// TIA Portal project "LabPLC" (V13)

(* hardware
DEVICE "S7-1200 station_1"  S7-1200 Station
   slot 0: "Rack_0"  Rack  V1.0
   slot 1: "LabPLC"  CPU 1215C DC/DC/DC  6ES7 215-1AG40-0XB0  V4.0
*)

// ===== PLC "LabPLC"  CPU 1215C DC/DC/DC =====

VAR_GLOBAL   // PLC tag table "Default tag table"
   "iTemp" AT %MW100 : Int;
   "PWM_Q1" AT %QW1002 : Int;
   "AxisFrequency_Pulse" AT %Q0.1 : Bool;
END_VAR

TYPE "User_data_type_1"
   STRUCT
      Notes : Array[0..15000] of Byte;
   END_STRUCT;
END_TYPE

DATA_BLOCK "dbInsMaster"   // DB2
{ S7_Optimized_Access := 'FALSE' }
VERSION : 0.1
// stored: InstanceOfName fbMaster
"fbMaster"
BEGIN
END_DATA_BLOCK

DATA_BLOCK "dbToneToFrequency"   // DB3
{ S7_Optimized_Access := 'FALSE' }
VERSION : 0.1
   VAR
      Freq : Array[0..128] of Int;
   END_VAR
BEGIN
   Freq[0] := 8;
   Freq[1] := 9;
   Freq[2] := 9;
   Freq[3] := 10;
   Freq[4] := 10;
   Freq[5] := 11;
   Freq[6] := 12;
   Freq[7] := 12;
   Freq[8] := 13;
   Freq[9] := 14;
   Freq[10] := 15;
   Freq[11] := 15;
   Freq[12] := 16;
   Freq[13] := 17;
   Freq[14] := 18;
   Freq[15] := 19;
   Freq[16] := 21;
   Freq[17] := 22;
   Freq[18] := 23;
   Freq[19] := 24;
   Freq[20] := 26;
   Freq[21] := 28;
   Freq[22] := 29;
   Freq[23] := 31;
   Freq[24] := 33;
   Freq[25] := 35;
   Freq[26] := 37;
   Freq[27] := 39;
   Freq[28] := 41;
   Freq[29] := 44;
   Freq[30] := 46;
   Freq[31] := 49;
   Freq[32] := 52;
   Freq[33] := 55;
   Freq[34] := 58;
   Freq[35] := 62;
   Freq[36] := 65;
   Freq[37] := 69;
   Freq[38] := 73;
   Freq[39] := 78;
   Freq[40] := 82;
   Freq[41] := 87;
   Freq[42] := 92;
   Freq[43] := 98;
   Freq[44] := 104;
   Freq[45] := 110;
   Freq[46] := 117;
   Freq[47] := 123;
   Freq[48] := 131;
   Freq[49] := 139;
   Freq[50] := 147;
   Freq[51] := 156;
   Freq[52] := 165;
   Freq[53] := 175;
   Freq[54] := 185;
   Freq[55] := 196;
   Freq[56] := 208;
   Freq[57] := 220;
   Freq[58] := 233;
   Freq[59] := 247;
   Freq[60] := 262;
   Freq[61] := 277;
   Freq[62] := 294;
   Freq[63] := 311;
   Freq[64] := 330;
   Freq[65] := 349;
   Freq[66] := 370;
   Freq[67] := 392;
   Freq[68] := 415;
   Freq[69] := 440;
   Freq[70] := 466;
   Freq[71] := 494;
   Freq[72] := 523;
   Freq[73] := 554;
   Freq[74] := 587;
   Freq[75] := 622;
   Freq[76] := 659;
   Freq[77] := 698;
   Freq[78] := 740;
   Freq[79] := 784;
   Freq[80] := 831;
   Freq[81] := 880;
   Freq[82] := 932;
   Freq[83] := 988;
   Freq[84] := 1047;
   Freq[85] := 1109;
   Freq[86] := 1175;
   Freq[87] := 1245;
   Freq[88] := 1319;
   Freq[89] := 1397;
   Freq[90] := 1480;
   Freq[91] := 1568;
   Freq[92] := 1661;
   Freq[93] := 1760;
   Freq[94] := 1865;
   Freq[95] := 1976;
   Freq[96] := 2093;
   Freq[97] := 2217;
   Freq[98] := 2349;
   Freq[99] := 2489;
   Freq[100] := 2637;
   Freq[101] := 2794;
   Freq[102] := 2960;
   Freq[103] := 3136;
   Freq[104] := 3322;
   Freq[105] := 3520;
   Freq[106] := 3729;
   Freq[107] := 3951;
   Freq[108] := 4186;
   Freq[109] := 4435;
   Freq[110] := 4699;
   Freq[111] := 4978;
   Freq[112] := 5274;
   Freq[113] := 5588;
   Freq[114] := 5920;
   Freq[115] := 6272;
   Freq[116] := 6645;
   Freq[117] := 7040;
   Freq[118] := 7459;
   Freq[119] := 7902;
   Freq[120] := 8372;
   Freq[121] := 8870;
   Freq[122] := 9397;
   Freq[123] := 9956;
   Freq[124] := 10548;
   Freq[125] := 11175;
   Freq[126] := 11840;
   Freq[127] := 12544;
   Freq[128] := 13290;
END_DATA_BLOCK

DATA_BLOCK "dbTunes"   // DB4
{ S7_Optimized_Access := 'FALSE' }
VERSION : 0.1
   VAR
      Tune_01 : Array[0..5000] of Byte;
   END_VAR
BEGIN
   Tune_01[0] := 0;
   Tune_01[1] := 36;
   Tune_01[2] := 16#0090;
   Tune_01[3] := 55;
   Tune_01[4] := 1;
   Tune_01[5] := 74;
   Tune_01[6] := 16#0080;
   Tune_01[7] := 0;
   Tune_01[8] := 242;
   Tune_01[9] := 16#0090;
   Tune_01[10] := 55;
   Tune_01[11] := 1;
   Tune_01[12] := 105;
   Tune_01[13] := 16#0080;
   Tune_01[14] := 0;
   Tune_01[15] := 232;
   Tune_01[16] := 16#0090;
   Tune_01[17] := 55;
   Tune_01[18] := 1;
   Tune_01[19] := 111;
   Tune_01[20] := 16#0080;
   Tune_01[21] := 0;
   Tune_01[22] := 202;
   Tune_01[23] := 16#0090;
   Tune_01[24] := 51;
   Tune_01[25] := 1;
   Tune_01[26] := 31;
   Tune_01[27] := 16#0080;
   Tune_01[28] := 0;
   Tune_01[29] := 147;
   Tune_01[30] := 16#0090;
   Tune_01[31] := 58;
   Tune_01[32] := 0;
   Tune_01[33] := 79;
   Tune_01[34] := 16#0080;
   Tune_01[35] := 0;
   Tune_01[36] := 69;
   Tune_01[37] := 16#0090;
   Tune_01[38] := 55;
   Tune_01[39] := 1;
   Tune_01[40] := 160;
   Tune_01[41] := 16#0080;
   Tune_01[42] := 0;
   Tune_01[43] := 165;
   Tune_01[44] := 16#0090;
   Tune_01[45] := 51;
   Tune_01[46] := 1;
   Tune_01[47] := 31;
   Tune_01[48] := 16#0080;
   Tune_01[49] := 0;
   Tune_01[50] := 169;
   Tune_01[51] := 16#0090;
   Tune_01[52] := 58;
   Tune_01[53] := 0;
   Tune_01[54] := 85;
   Tune_01[55] := 16#0080;
   Tune_01[56] := 0;
   Tune_01[57] := 51;
   Tune_01[58] := 16#0090;
   Tune_01[59] := 55;
   Tune_01[60] := 2;
   Tune_01[61] := 235;
   Tune_01[62] := 16#0080;
   Tune_01[63] := 1;
   Tune_01[64] := 166;
   Tune_01[65] := 16#0090;
   Tune_01[66] := 62;
   Tune_01[67] := 1;
   Tune_01[68] := 121;
   Tune_01[69] := 16#0080;
   Tune_01[70] := 0;
   Tune_01[71] := 216;
   Tune_01[72] := 16#0090;
   Tune_01[73] := 62;
   Tune_01[74] := 1;
   Tune_01[75] := 115;
   Tune_01[76] := 16#0080;
   Tune_01[77] := 0;
   Tune_01[78] := 208;
   Tune_01[79] := 16#0090;
   Tune_01[80] := 62;
   Tune_01[81] := 1;
   Tune_01[82] := 130;
   Tune_01[83] := 16#0080;
   Tune_01[84] := 0;
   Tune_01[85] := 223;
   Tune_01[86] := 16#0090;
   Tune_01[87] := 63;
   Tune_01[88] := 1;
   Tune_01[89] := 1;
   Tune_01[90] := 16#0080;
   Tune_01[91] := 0;
   Tune_01[92] := 165;
   Tune_01[93] := 16#0090;
   Tune_01[94] := 58;
   Tune_01[95] := 0;
   Tune_01[96] := 95;
   Tune_01[97] := 16#0080;
   Tune_01[98] := 0;
   Tune_01[99] := 69;
   Tune_01[100] := 16#0090;
   Tune_01[101] := 54;
   Tune_01[102] := 1;
   Tune_01[103] := 160;
   Tune_01[104] := 16#0080;
   Tune_01[105] := 0;
   Tune_01[106] := 156;
   Tune_01[107] := 16#0090;
   Tune_01[108] := 51;
   Tune_01[109] := 0;
   Tune_01[110] := 248;
   Tune_01[111] := 16#0080;
   Tune_01[112] := 0;
   Tune_01[113] := 176;
   Tune_01[114] := 16#0090;
   Tune_01[115] := 58;
   Tune_01[116] := 0;
   Tune_01[117] := 85;
   Tune_01[118] := 16#0080;
   Tune_01[119] := 0;
   Tune_01[120] := 79;
   Tune_01[121] := 16#0090;
   Tune_01[122] := 55;
   Tune_01[123] := 2;
   Tune_01[124] := 2;
   Tune_01[125] := 16#0080;
   Tune_01[126] := 2;
   Tune_01[127] := 143;
   Tune_01[128] := 16#0090;
   Tune_01[129] := 67;
   Tune_01[130] := 1;
   Tune_01[131] := 201;
   Tune_01[132] := 16#0080;
   Tune_01[133] := 0;
   Tune_01[134] := 131;
   Tune_01[135] := 16#0090;
   Tune_01[136] := 55;
   Tune_01[137] := 1;
   Tune_01[138] := 41;
   Tune_01[139] := 16#0080;
   Tune_01[140] := 0;
   Tune_01[141] := 161;
   Tune_01[142] := 16#0090;
   Tune_01[143] := 55;
   Tune_01[144] := 0;
   Tune_01[145] := 116;
   Tune_01[146] := 16#0080;
   Tune_01[147] := 0;
   Tune_01[148] := 34;
   Tune_01[149] := 16#0090;
   Tune_01[150] := 67;
   Tune_01[151] := 1;
   Tune_01[152] := 115;
   Tune_01[153] := 16#0080;
   Tune_01[154] := 0;
   Tune_01[155] := 164;
   Tune_01[156] := 16#0090;
   Tune_01[157] := 66;
   Tune_01[158] := 1;
   Tune_01[159] := 62;
   Tune_01[160] := 16#0080;
   Tune_01[161] := 0;
   Tune_01[162] := 153;
   Tune_01[163] := 16#0090;
   Tune_01[164] := 65;
   Tune_01[165] := 0;
   Tune_01[166] := 98;
   Tune_01[167] := 16#0080;
   Tune_01[168] := 0;
   Tune_01[169] := 49;
   Tune_01[170] := 16#0090;
   Tune_01[171] := 64;
   Tune_01[172] := 0;
   Tune_01[173] := 140;
   Tune_01[174] := 16#0080;
   Tune_01[175] := 0;
   Tune_01[176] := 6;
   Tune_01[177] := 16#0090;
   Tune_01[178] := 63;
   Tune_01[179] := 0;
   Tune_01[180] := 101;
   Tune_01[181] := 16#0080;
   Tune_01[182] := 0;
   Tune_01[183] := 45;
   Tune_01[184] := 16#0090;
   Tune_01[185] := 64;
   Tune_01[186] := 0;
   Tune_01[187] := 132;
   Tune_01[188] := 16#0080;
   Tune_01[189] := 1;
   Tune_01[190] := 212;
   Tune_01[191] := 16#0090;
   Tune_01[192] := 56;
   Tune_01[193] := 0;
   Tune_01[194] := 113;
   Tune_01[195] := 16#0080;
   Tune_01[196] := 0;
   Tune_01[197] := 183;
   Tune_01[198] := 16#0090;
   Tune_01[199] := 61;
   Tune_01[200] := 1;
   Tune_01[201] := 133;
   Tune_01[202] := 16#0080;
   Tune_01[203] := 0;
   Tune_01[204] := 198;
   Tune_01[205] := 16#0090;
   Tune_01[206] := 60;
   Tune_01[207] := 1;
   Tune_01[208] := 66;
   Tune_01[209] := 16#0080;
   Tune_01[210] := 0;
   Tune_01[211] := 118;
   Tune_01[212] := 16#0090;
   Tune_01[213] := 59;
   Tune_01[214] := 0;
   Tune_01[215] := 107;
   Tune_01[216] := 16#0080;
   Tune_01[217] := 0;
   Tune_01[218] := 45;
   Tune_01[219] := 16#0090;
   Tune_01[220] := 58;
   Tune_01[221] := 0;
   Tune_01[222] := 113;
   Tune_01[223] := 16#0080;
   Tune_01[224] := 0;
   Tune_01[225] := 20;
   Tune_01[226] := 16#0090;
   Tune_01[227] := 57;
   Tune_01[228] := 0;
   Tune_01[229] := 89;
   Tune_01[230] := 16#0080;
   Tune_01[231] := 0;
   Tune_01[232] := 60;
   Tune_01[233] := 16#0090;
   Tune_01[234] := 58;
   Tune_01[235] := 0;
   Tune_01[236] := 128;
   Tune_01[237] := 16#0080;
   Tune_01[238] := 1;
   Tune_01[239] := 213;
   Tune_01[240] := 16#0090;
   Tune_01[241] := 51;
   Tune_01[242] := 0;
   Tune_01[243] := 98;
   Tune_01[244] := 16#0080;
   Tune_01[245] := 0;
   Tune_01[246] := 192;
   Tune_01[247] := 16#0090;
   Tune_01[248] := 54;
   Tune_01[249] := 1;
   Tune_01[250] := 99;
   Tune_01[251] := 16#0080;
   Tune_01[252] := 0;
   Tune_01[253] := 245;
   Tune_01[254] := 16#0090;
   Tune_01[255] := 51;
   Tune_01[256] := 1;
   Tune_01[257] := 81;
   Tune_01[258] := 16#0080;
   Tune_01[259] := 0;
   Tune_01[260] := 104;
   Tune_01[261] := 16#0090;
   Tune_01[262] := 54;
   Tune_01[263] := 0;
   Tune_01[264] := 73;
   Tune_01[265] := 16#0080;
   Tune_01[266] := 0;
   Tune_01[267] := 89;
   Tune_01[268] := 16#0090;
   Tune_01[269] := 58;
   Tune_01[270] := 1;
   Tune_01[271] := 139;
   Tune_01[272] := 16#0080;
   Tune_01[273] := 0;
   Tune_01[274] := 164;
   Tune_01[275] := 16#0090;
   Tune_01[276] := 55;
   Tune_01[277] := 1;
   Tune_01[278] := 74;
   Tune_01[279] := 16#0080;
   Tune_01[280] := 0;
   Tune_01[281] := 110;
   Tune_01[282] := 16#0090;
   Tune_01[283] := 58;
   Tune_01[284] := 0;
   Tune_01[285] := 79;
   Tune_01[286] := 16#0080;
   Tune_01[287] := 0;
   Tune_01[288] := 79;
   Tune_01[289] := 16#0090;
   Tune_01[290] := 62;
   Tune_01[291] := 2;
   Tune_01[292] := 233;
   Tune_01[293] := 16#0080;
   Tune_01[294] := 1;
   Tune_01[295] := 144;
   Tune_01[296] := 16#0090;
   Tune_01[297] := 67;
   Tune_01[298] := 1;
   Tune_01[299] := 201;
   Tune_01[300] := 16#0080;
   Tune_01[301] := 0;
   Tune_01[302] := 131;
   Tune_01[303] := 16#0090;
   Tune_01[304] := 55;
   Tune_01[305] := 1;
   Tune_01[306] := 41;
   Tune_01[307] := 16#0080;
   Tune_01[308] := 0;
   Tune_01[309] := 161;
   Tune_01[310] := 16#0090;
   Tune_01[311] := 55;
   Tune_01[312] := 0;
   Tune_01[313] := 116;
   Tune_01[314] := 16#0080;
   Tune_01[315] := 0;
   Tune_01[316] := 34;
   Tune_01[317] := 16#0090;
   Tune_01[318] := 67;
   Tune_01[319] := 1;
   Tune_01[320] := 115;
   Tune_01[321] := 16#0080;
   Tune_01[322] := 0;
   Tune_01[323] := 164;
   Tune_01[324] := 16#0090;
   Tune_01[325] := 66;
   Tune_01[326] := 1;
   Tune_01[327] := 62;
   Tune_01[328] := 16#0080;
   Tune_01[329] := 0;
   Tune_01[330] := 153;
   Tune_01[331] := 16#0090;
   Tune_01[332] := 65;
   Tune_01[333] := 0;
   Tune_01[334] := 98;
   Tune_01[335] := 16#0080;
   Tune_01[336] := 0;
   Tune_01[337] := 49;
   Tune_01[338] := 16#0090;
   Tune_01[339] := 64;
   Tune_01[340] := 0;
   Tune_01[341] := 140;
   Tune_01[342] := 16#0080;
   Tune_01[343] := 0;
   Tune_01[344] := 6;
   Tune_01[345] := 16#0090;
   Tune_01[346] := 63;
   Tune_01[347] := 0;
   Tune_01[348] := 101;
   Tune_01[349] := 16#0080;
   Tune_01[350] := 0;
   Tune_01[351] := 45;
   Tune_01[352] := 16#0090;
   Tune_01[353] := 64;
   Tune_01[354] := 0;
   Tune_01[355] := 132;
   Tune_01[356] := 16#0080;
   Tune_01[357] := 1;
   Tune_01[358] := 212;
   Tune_01[359] := 16#0090;
   Tune_01[360] := 56;
   Tune_01[361] := 0;
   Tune_01[362] := 113;
   Tune_01[363] := 16#0080;
   Tune_01[364] := 0;
   Tune_01[365] := 183;
   Tune_01[366] := 16#0090;
   Tune_01[367] := 61;
   Tune_01[368] := 1;
   Tune_01[369] := 133;
   Tune_01[370] := 16#0080;
   Tune_01[371] := 0;
   Tune_01[372] := 198;
   Tune_01[373] := 16#0090;
   Tune_01[374] := 60;
   Tune_01[375] := 1;
   Tune_01[376] := 66;
   Tune_01[377] := 16#0080;
   Tune_01[378] := 0;
   Tune_01[379] := 118;
   Tune_01[380] := 16#0090;
   Tune_01[381] := 59;
   Tune_01[382] := 0;
   Tune_01[383] := 83;
   Tune_01[384] := 16#0080;
   Tune_01[385] := 0;
   Tune_01[386] := 57;
   Tune_01[387] := 16#0090;
   Tune_01[388] := 58;
   Tune_01[389] := 0;
   Tune_01[390] := 113;
   Tune_01[391] := 16#0080;
   Tune_01[392] := 0;
   Tune_01[393] := 26;
   Tune_01[394] := 16#0090;
   Tune_01[395] := 57;
   Tune_01[396] := 0;
   Tune_01[397] := 89;
   Tune_01[398] := 16#0080;
   Tune_01[399] := 0;
   Tune_01[400] := 60;
   Tune_01[401] := 16#0090;
   Tune_01[402] := 58;
   Tune_01[403] := 0;
   Tune_01[404] := 128;
   Tune_01[405] := 16#0080;
   Tune_01[406] := 1;
   Tune_01[407] := 219;
   Tune_01[408] := 16#0090;
   Tune_01[409] := 51;
   Tune_01[410] := 0;
   Tune_01[411] := 98;
   Tune_01[412] := 16#0080;
   Tune_01[413] := 0;
   Tune_01[414] := 192;
   Tune_01[415] := 16#0090;
   Tune_01[416] := 54;
   Tune_01[417] := 1;
   Tune_01[418] := 99;
   Tune_01[419] := 16#0080;
   Tune_01[420] := 0;
   Tune_01[421] := 230;
   Tune_01[422] := 16#0090;
   Tune_01[423] := 51;
   Tune_01[424] := 1;
   Tune_01[425] := 81;
   Tune_01[426] := 16#0080;
   Tune_01[427] := 0;
   Tune_01[428] := 116;
   Tune_01[429] := 16#0090;
   Tune_01[430] := 58;
   Tune_01[431] := 0;
   Tune_01[432] := 73;
   Tune_01[433] := 16#0080;
   Tune_01[434] := 0;
   Tune_01[435] := 61;
   Tune_01[436] := 16#0090;
   Tune_01[437] := 55;
   Tune_01[438] := 1;
   Tune_01[439] := 142;
   Tune_01[440] := 16#0080;
   Tune_01[441] := 0;
   Tune_01[442] := 177;
   Tune_01[443] := 16#0090;
   Tune_01[444] := 51;
   Tune_01[445] := 1;
   Tune_01[446] := 74;
   Tune_01[447] := 16#0080;
   Tune_01[448] := 0;
   Tune_01[449] := 140;
   Tune_01[450] := 16#0090;
   Tune_01[451] := 58;
   Tune_01[452] := 0;
   Tune_01[453] := 79;
   Tune_01[454] := 16#0080;
   Tune_01[455] := 0;
   Tune_01[456] := 49;
   Tune_01[457] := 16#0090;
   Tune_01[458] := 55;
   Tune_01[459] := 2;
   Tune_01[460] := 229;
   Tune_01[461] := 16#0080;
   Tune_01[462] := 16#00F0;
   Tune_01[463] := 177;
   Tune_01[464] := 16#0090;
   Tune_01[465] := 51;
   Tune_01[466] := 1;
   Tune_01[467] := 74;
   Tune_01[468] := 16#0080;
   Tune_01[469] := 0;
   Tune_01[470] := 140;
   Tune_01[471] := 16#0090;
   Tune_01[472] := 58;
   Tune_01[473] := 0;
   Tune_01[474] := 79;
   Tune_01[475] := 16#0080;
   Tune_01[476] := 0;
   Tune_01[477] := 49;
   Tune_01[478] := 16#0090;
   Tune_01[479] := 55;
   Tune_01[480] := 2;
   Tune_01[481] := 229;
   Tune_01[482] := 16#0080;
END_DATA_BLOCK

DATA_BLOCK "AxisFrequency"   // DB1, Motion_DB
{ S7_Optimized_Access := 'FALSE' }
AUTHOR : SIMATIC
FAMILY : BasicMC
NAME : TO_PosAx
VERSION : 4.0
// stored: InstanceOfName ?
"?"
BEGIN
END_DATA_BLOCK

FUNCTION_BLOCK "fbMaster"   // FB1, LAD
{ S7_Optimized_Access := 'FALSE' }
VERSION : 0.1
   VAR
      MV_Frequency : MC_MoveVelocity;
      MP_Frequency : MC_Power;
      MID_MidiParser : "fbMidi";
      rPrevFrequency : Real;
      rFrequency : Real;
   END_VAR
   VAR_TEMP
      bTemp : Bool;
      wTemp : Word;
      iTemp : Int;
      rTemp : Real;
   END_VAR
   VAR_TEMP   // added for the SCL form of the ladder/FBD networks
      _w1 : Bool;
   END_VAR
BEGIN

REGION Network 1
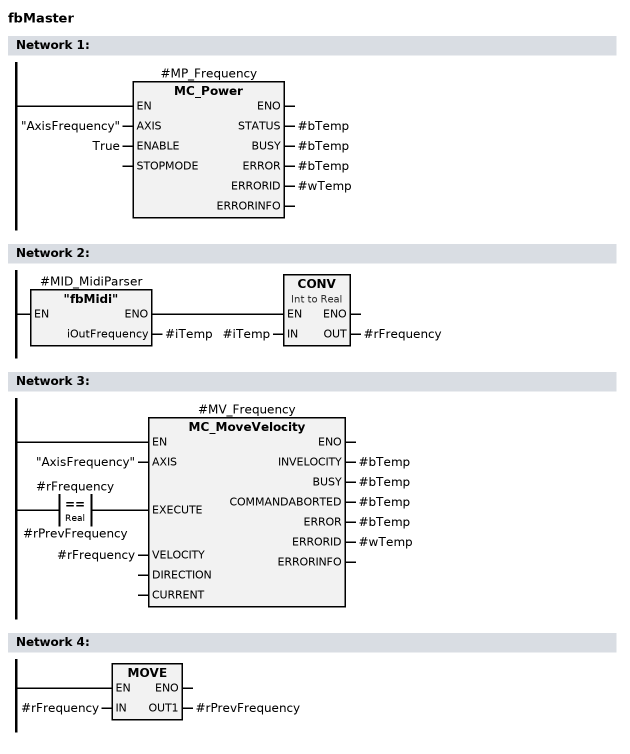
   #MP_Frequency(Axis := "AxisFrequency",   // MC_Power
                 Enable := True,
                 Status => #bTemp,
                 Busy => #bTemp,
                 Error => #bTemp,
                 ErrorID => #wTemp);
END_REGION

REGION Network 2
   RUNG wire#powerrail
      #MID_MidiParser(iOutFrequency => #iTemp)
      { S7_Templates := "[SrcType := Int, DestType := Real]" } Convert(in := #iTemp, out => #rFrequency)
   END_RUNG
   // the same network as SCL:
   #MID_MidiParser(iOutFrequency => #iTemp, ENO => #_w1);   // "fbMidi"
   IF #_w1 THEN #rFrequency := INT_TO_REAL(#iTemp); END_IF;
END_REGION

REGION Network 3
   #MV_Frequency(Axis := "AxisFrequency",   // MC_MoveVelocity
                 Execute := #rFrequency = #rPrevFrequency,
                 Velocity := #rFrequency,
                 InVelocity => #bTemp,
                 Busy => #bTemp,
                 CommandAborted => #bTemp,
                 Error => #bTemp,
                 ErrorID => #wTemp);
END_REGION

REGION Network 4
   RUNG wire#powerrail
      Move(in := #rFrequency, out1 => #rPrevFrequency)
   END_RUNG
   // the same network as SCL:
   #rPrevFrequency := #rFrequency;
END_REGION
END_FUNCTION_BLOCK

FUNCTION_BLOCK "fbMidi"   // FB2, SCL
{ S7_Optimized_Access := 'FALSE' }
VERSION : 0.1
   VAR_OUTPUT
      iOutFrequency : Int;
   END_VAR
   VAR
      TON_Delay : TON_TIME;
      byCmd : Byte;
      iDelay : Int;
      byOpCode : Byte;
      byNote : Byte;
      bDelayRunning : Bool;
      iCursor : Int;
   END_VAR
BEGIN
   // Be sure we not waiting for delay to complete
   IF NOT #bDelayRunning OR (#bDelayRunning AND #TON_Delay.Q) THEN
       // Reset delay bit
       #bDelayRunning := false;

       // Read midi commad
       #byCmd := "dbTunes".Tune_01[#iCursor];
       #iCursor := #iCursor + 1;

       // Delay command?
       IF #byCmd < 16#80 THEN
           // Wait
           #iDelay := SHL(IN := BYTE_TO_WORD(#byCmd), N := 8) + "dbTunes".Tune_01[#iCursor];
           #iCursor := #iCursor + 1;
           #bDelayRunning := true;
       END_IF;

       // Get opcode
       #byOpCode := #byCmd AND 16#F0;
       CASE BYTE_TO_INT(#byOpCode) OF
           16#80:
               // Stop note
               #iOutFrequency := 0;

          16#90:
               // Start note
               #byNote := "dbTunes".Tune_01[#iCursor];
               #iCursor := #iCursor + 1;

               IF #byNote > 127 THEN
                   #byNote := 127;
               END_IF;
               #iOutFrequency := "dbToneToFrequency".Freq[#byNote];

           16#E0:
               // Restart
               #iCursor := 0;

           16#F0:
               // Stop
               #iCursor := 0;
       END_CASE;
   END_IF;

   // Delay ms if needed
   #TON_Delay(IN := #bDelayRunning, PT := INT_TO_TIME(#iDelay));
END_FUNCTION_BLOCK

ORGANIZATION_BLOCK "Main"   // OB1, LAD, ProgramCycle
TITLE = "Main Program Sweep (Cycle)"
{ S7_Optimized_Access := 'FALSE' }
VERSION : 0.1
   VAR_INPUT
      Initial_Call : Bool;   // Initial call of this OB
      Remanence : Bool;   // =True, if remanent data are available
   END_VAR
BEGIN

REGION Network 1
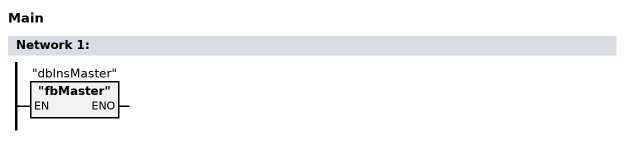
   RUNG wire#powerrail
      "dbInsMaster"()
   END_RUNG
   // the same network as SCL:
   "dbInsMaster"();   // "fbMaster"
END_REGION
END_ORGANIZATION_BLOCK